# EPICS substitutions: Initial/db/user.substitutions
# Example substitutions file

file "db/dbExample1.db" {
    { user = "hbui" }
}

file "db/dbExample2.db" {
    pattern { user, no, scan }
        { "hbui", 1, "1 second" }
        { "hbui", 2, "2 second" }
        { "hbui", 3, "5 second" }
}
